{attribute addProperty BoxType "EP7402-0057-0017"}
{attribute addProperty Id "VelocityAT %Q*INT16233AccellerationAT %Q*UINT16234DeccelerationAT %Q*UINT16235"}
{attribute addProperty CRC "1089323787"}
{attribute addProperty SizeInBites "48"}
{attribute addProperty SizeInBytes "6"}
TYPE STM_Target_Velocity_Channel_40EDC30B :
STRUCT
	{attribute addProperty Name "Velocity"}
	Velocity AT %Q* : INT;
	{attribute addProperty Name "Accelleration"}
	Accelleration AT %Q* : UINT;
	{attribute addProperty Name "Decceleration"}
	Decceleration AT %Q* : UINT;
END_STRUCT
END_TYPE

(* stored: Version 1.2.0.0, ProductVersion 3.1.4024.9
   DUT STM_Target_Velocity_Channel_40EDC30B: Id {fd67e9e0-859d-4e57-b037-f83254552f20} *)
